// Checks if a string is a signed interger
FUNCTION F_ISSIGNEDINT : BOOL
VAR_INPUT
	sValue : REFERENCE TO STRING;
END_VAR
VAR
	i : T_Size;
END_VAR

F_TRIMWHITESPACE(sValue, T_Whitespace_Location.Both);

IF F_BYTETOCHAR(sValue[0]) = '+' OR_ELSE F_BYTETOCHAR(sValue[0]) = '-' THEN i := i + 1; END_IF
IF NOT F_ISDIGIT(F_BYTETOCHAR(sValue[i])) THEN RETURN; END_IF
WHILE F_ISDIGIT(F_BYTETOCHAR(sValue[i])) DO i := i + 1; END_WHILE
F_ISSIGNEDINT := sValue[i] = 0;

END_FUNCTION

(* stored: Version 1.1.0.1, ProductVersion 3.1.4024.4
   POU F_ISSIGNEDINT: Id {53f0e721-cef1-4e7f-9775-68c2ea9fe311}, SpecialFunc None *)
